Universal Robots PolyScope program: screwdriver.urp

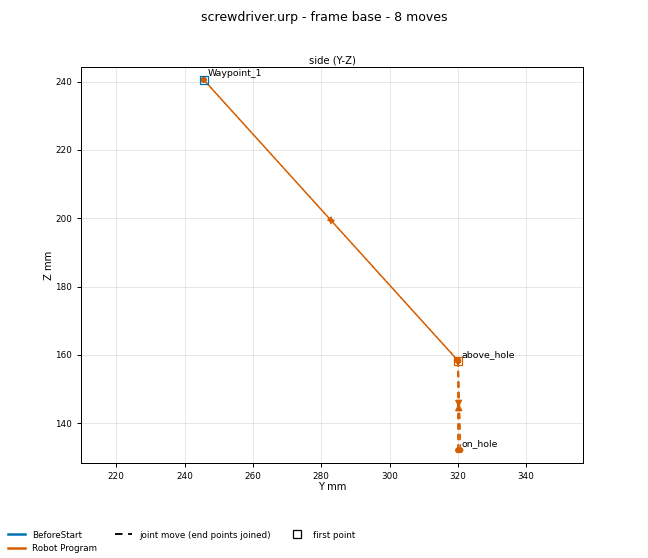
[picture p0: tool path of screwdriver.urp in frame base, 8 of 8 moves have a stored position in this frame; points joined in program order, loops and branches not executed]
Program Argonne labs (installation=default directory=/programs/AlexT/Argonne labs createdIn=5.13.0 lastSavedIn=5.13.0 robotSerialNumber=20185501097)
Calibrated DH parameters: a=[0.000228, -0.136104, -0.213225, -0.000132, 0.000212, 0]; d=[0.162425, 140.257984, -310.855376, 170.730986, 0.099888, 0.099591]; alpha=[1.569577, -0.002871, 0.001929, 1.574027, -1.569315, 0]; deltaTheta=[0, -1.244856, 0.248959, 0.995903, -0.000001, 0]
InitVariablesNode
BeforeStart
  MoveJ speed 60 deg/s, acceleration 80 deg/s^2 (useActiveTCP=true) feature=Base
    Waypoint Waypoint_1: TCP in base x=335.641 y=245.606 z=240.509 mm, rx=-3.1412 ry=0 rz=-0.0003 rad; joints [201.601, -111.658, 104.049, -82.322, -89.843, -68.691] deg; TCP offset x=76 y=0 z=269 mm, rx=0 ry=0 rz=0 rad
Robot Program (runOnlyOnce=false)
  Script: rq_screw_vacuum_on()
  Popup Message (haltProgram=false message=Add insert inputType=Text)
  MoveJ speed 60 deg/s, acceleration 80 deg/s^2 (useActiveTCP=true) feature=Base
    Waypoint above_hole: TCP in base x=335.649 y=320.063 z=158.27 mm, rx=-3.1412 ry=0 rz=-0.0003 rad; joints [212.153, -103.457, 110.577, -97.057, -89.822, -58.1] deg
    Waypoint on_hole: TCP in base x=335.681 y=320.034 z=132.086 mm, rx=-3.1412 ry=0.0001 rz=-0.0004 rad; joints [212.152, -102.851, 113.999, -101.089, -89.818, -58.091] deg
    URCap Drive Screw (Robotiq_Screwdriving, Robotiq Inc.) dataModel(selectedStopConditionKey=2, metricTorqueStopConditionKey={"value":0.3,"type":"METRIC_TORQUE"}, toolSpeedKey=100, advancedSettingsVisibleKey=true, threadMatingPositionKey=p[0.3358571246996078, 0.3200813392125644, 0.1318888242204277, -3.14088180381315, 1.4901171715672826E-4, -0.001505484901946036], finalPositionKey=p[0.33574183730424734, 0.3200829252058823, 0.12663880454164606, -3.1408982631825952, 1.701079722584559E-4, -9.392136887126088E-4], degreesBeforeRampDownKey=1197, torqueThresholdKey=2152, torqueAngleSlopeKey=1403)
      URCap Robotiq Folder Node (Robotiq_Screwdriving, Robotiq Inc.) dataModel(TitleKey=If success)
        'Insert If Success Instructions'
        MoveL speed 250 mm/s, acceleration 1200 mm/s^2 (useActiveTCP=true) feature=Base
          MoveDirectionNode (selectedDirection=ZMinus) feature=Joint_6_name
            Until DISTANCE (allowActions=false deceleration=3 distanceNodeType=STOP) Distance=0.005; motionParameters(blendRadius=0)
      URCap Robotiq Folder Node (Robotiq_Screwdriving, Robotiq Inc.) dataModel(TitleKey=If fail)
        URCap Robotiq Folder Node (Robotiq_Screwdriving, Robotiq Inc.) dataModel(TitleKey=No screw detected)
          Popup Error (haltProgram=false message=No screw detected inputType=Text)
        URCap Robotiq Folder Node (Robotiq_Screwdriving, Robotiq Inc.) dataModel(TitleKey=Timeout reached)
          Popup Error (haltProgram=false message=Timeout reached inputType=Text)
        URCap Robotiq Folder Node (Robotiq_Screwdriving, Robotiq Inc.) dataModel(TitleKey=Screwdriver not activated)
          Popup Error (haltProgram=false message=Screwdriver Not Activated inputType=Text)
        URCap Robotiq Folder Node (Robotiq_Screwdriving, Robotiq Inc.) dataModel(TitleKey=Unhandled errors)
          Popup Error (haltProgram=false message=Unhandled Screwdriving Error: Open Log tab for information on application warnings, and refer to the Screwdriver instruction manual to manage faults. inputType=Text)
  MoveJ speed 60 deg/s, acceleration 80 deg/s^2 (useActiveTCP=true) feature=Base
    Waypoint above_hole: TCP in base x=335.649 y=320.063 z=158.27 mm, rx=-3.1412 ry=0 rz=-0.0003 rad; joints [212.153, -103.457, 110.577, -97.057, -89.822, -58.1] deg
    Waypoint Waypoint_1: TCP in base x=335.641 y=245.606 z=240.509 mm, rx=-3.1412 ry=0 rz=-0.0003 rad; joints [201.601, -111.658, 104.049, -82.322, -89.843, -68.691] deg
    Script: rq_screw_vacuum_on()
  Popup Message (haltProgram=false message=Flip part and add new insert. inputType=Text)
  MoveJ speed 60 deg/s, acceleration 80 deg/s^2 (useActiveTCP=true) feature=Base
    Waypoint above_hole: TCP in base x=335.649 y=320.063 z=158.27 mm, rx=-3.1412 ry=0 rz=-0.0003 rad; joints [212.153, -103.457, 110.577, -97.057, -89.822, -58.1] deg
    Waypoint on_hole_2: TCP in base x=335.878 y=320.732 z=132.106 mm, rx=-3.1412 ry=0.0001 rz=-0.0004 rad; joints [212.224, -102.746, 113.915, -101.105, -89.819, -58.019] deg
  URCap Drive Screw (Robotiq_Screwdriving, Robotiq Inc.) dataModel(selectedStopConditionKey=2, metricTorqueStopConditionKey={"value":0.3,"type":"METRIC_TORQUE"}, toolSpeedKey=100, advancedSettingsVisibleKey=true, threadMatingPositionKey=p[0.3358571246996078, 0.3200813392125644, 0.1318888242204277, -3.14088180381315, 1.4901171715672826E-4, -0.001505484901946036], finalPositionKey=p[0.33574183730424734, 0.3200829252058823, 0.12663880454164606, -3.1408982631825952, 1.701079722584559E-4, -9.392136887126088E-4], degreesBeforeRampDownKey=1197, torqueThresholdKey=2152, torqueAngleSlopeKey=1403)
    URCap Robotiq Folder Node (Robotiq_Screwdriving, Robotiq Inc.) dataModel(TitleKey=If success)
      'Insert If Success Instructions'
      MoveL speed 250 mm/s, acceleration 1200 mm/s^2 (useActiveTCP=true) feature=Base
        MoveDirectionNode (selectedDirection=ZMinus) feature=Joint_6_name
          Until DISTANCE (allowActions=false deceleration=3 distanceNodeType=STOP) Distance=0.005; motionParameters(blendRadius=0)
    URCap Robotiq Folder Node (Robotiq_Screwdriving, Robotiq Inc.) dataModel(TitleKey=If fail)
      URCap Robotiq Folder Node (Robotiq_Screwdriving, Robotiq Inc.) dataModel(TitleKey=No screw detected)
        Popup Error (haltProgram=false message=No screw detected inputType=Text)
      URCap Robotiq Folder Node (Robotiq_Screwdriving, Robotiq Inc.) dataModel(TitleKey=Timeout reached)
        Popup Error (haltProgram=false message=Timeout reached inputType=Text)
      URCap Robotiq Folder Node (Robotiq_Screwdriving, Robotiq Inc.) dataModel(TitleKey=Screwdriver not activated)
        Popup Error (haltProgram=false message=Screwdriver Not Activated inputType=Text)
      URCap Robotiq Folder Node (Robotiq_Screwdriving, Robotiq Inc.) dataModel(TitleKey=Unhandled errors)
        Popup Error (haltProgram=false message=Unhandled Screwdriving Error: Open Log tab for information on application warnings, and refer to the Screwdriver instruction manual to manage faults. inputType=Text)
  MoveJ speed 60 deg/s, acceleration 80 deg/s^2 (useActiveTCP=true) feature=Base
    Waypoint above_hole: TCP in base x=335.649 y=320.063 z=158.27 mm, rx=-3.1412 ry=0 rz=-0.0003 rad; joints [212.153, -103.457, 110.577, -97.057, -89.822, -58.1] deg
  Halt
